// TIA Portal V17 export
// export: Created 2025-06-26T07:49:12.8762172Z, ExportSetting WithDefaults, DisplayName Totally Integrated Automation Portal, DisplayVersion V17 Update 8, DisplayName TIA Portal Openness, DisplayVersion V17 Update 8, DisplayName TIA Portal Version Control Interface, DisplayVersion V17, DisplayName STEP 7 Professional, DisplayVersion V17 Update 8, DisplayName STEP 7 Safety, DisplayVersion V17 Update 6, DisplayName WinCC Advanced, DisplayVersion V17 Update 8
ORGANIZATION_BLOCK "CAN_CyclicInterrupt"   // OB30, FBD, CyclicInterrupt
{ S7_Optimized_Access := 'TRUE' }
VERSION : 0.1
// stored: AutoNumber true, IsIECCheckEnabled false, SetENOAutomatically false
   VAR_INPUT
      Initial_Call : Bool;   // Initial call of this OB
      Event_Count : Int;   // Events discarded
   END_VAR
BEGIN

REGION Network 1: CAN communication
   // EN := "DB_CurrentSetting"."CAN-Module_Active"
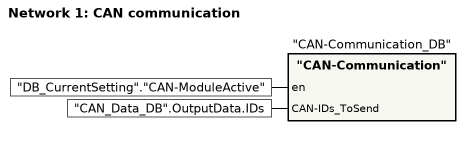
   IF "DB_CurrentSetting"."CAN-ModuleActive" THEN
       "CAN-Communication_DB"("CAN-IDs_ToSend" := "CAN_Data_DB".OutputData.IDs);   // "CAN-Communication"
   END_IF;
END_REGION
END_ORGANIZATION_BLOCK
